// TIA Portal V19 export
TYPE "C402_STU_M33_TYPIC"
   STRUCT
      CMD { ExternalAccessible := 'False'; ExternalVisible := 'False'; ExternalWritable := 'False'} : Bool;   // Sturing M33-bord
   END_STRUCT;
END_TYPE
